# EPICS autosave request: support/ip-2-10/ipApp/Db/Agilent_E3631A_settings.req
#FILE... Agilent_E3631A_settings.req
#USAGE... Agilent_E3631A.db fields autosave'd.
$(P)E3631A:$(S):setV_P6V
$(P)E3631A:$(S):setC_P6V
$(P)E3631A:$(S):setV_P25V
$(P)E3631A:$(S):setC_P25V
$(P)E3631A:$(S):setV_N25V
$(P)E3631A:$(S):setC_N25V
$(P)E3631A:$(S):locRem
$(P)E3631A:$(S):output
